// TIA Portal V18 export
FUNCTION "Scale" : Void   // FC2, LAD
{ S7_Optimized_Access := 'TRUE' }
VERSION : 0.1
// stored: AutoNumber true, IsIECCheckEnabled false, SetENOAutomatically false, UDAEnableTagReadback false
   VAR_TEMP
      temp : Real;
   END_VAR
BEGIN

REGION Network 1: Flow meter
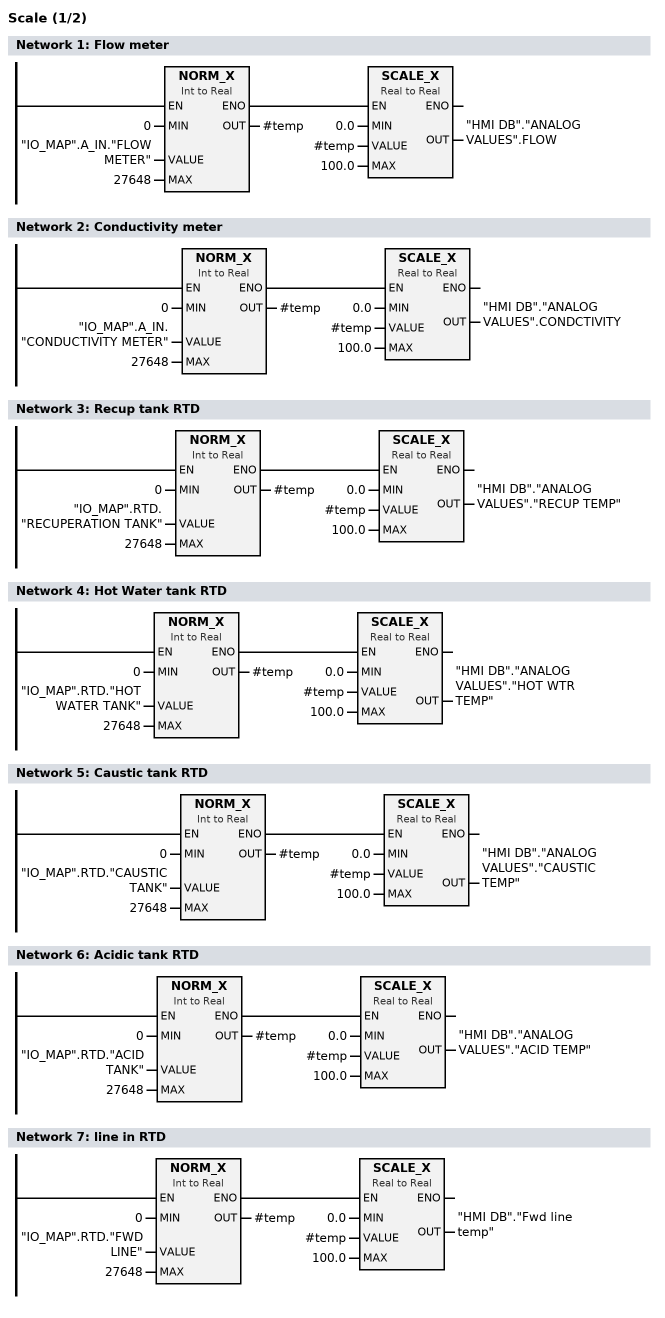
   RUNG wire#powerrail
      { S7_Templates := "[SrcType := Int, DestType := Real]" } Normalize(min := 0, value := "IO_MAP".A_IN."FLOW METER", max := 27648, out => #temp)
      { S7_Templates := "[SrcType := Real, DestType := Real]" } Scale(min := 0.0, value := #temp, max := 100.0, out => "HMI DB"."ANALOG VALUES".FLOW)
   END_RUNG
   // the same network as SCL:
   #temp := NORM_X(MIN := 0, VALUE := "IO_MAP".A_IN."FLOW METER", MAX := 27648);
   "HMI DB"."ANALOG VALUES".FLOW := SCALE_X(MIN := 0.0, VALUE := #temp, MAX := 100.0);
END_REGION

REGION Network 2: Conductivity meter
   RUNG wire#powerrail
      { S7_Templates := "[SrcType := Int, DestType := Real]" } Normalize(min := 0, value := "IO_MAP".A_IN."CONDUCTIVITY METER", max := 27648, out => #temp)
      { S7_Templates := "[SrcType := Real, DestType := Real]" } Scale(min := 0.0, value := #temp, max := 100.0, out => "HMI DB"."ANALOG VALUES".CONDCTIVITY)
   END_RUNG
   // the same network as SCL:
   #temp := NORM_X(MIN := 0, VALUE := "IO_MAP".A_IN."CONDUCTIVITY METER", MAX := 27648);
   "HMI DB"."ANALOG VALUES".CONDCTIVITY := SCALE_X(MIN := 0.0, VALUE := #temp, MAX := 100.0);
END_REGION

REGION Network 3: Recup tank RTD
   RUNG wire#powerrail
      { S7_Templates := "[SrcType := Int, DestType := Real]" } Normalize(min := 0, value := "IO_MAP".RTD."RECUPERATION TANK", max := 27648, out => #temp)
      { S7_Templates := "[SrcType := Real, DestType := Real]" } Scale(min := 0.0, value := #temp, max := 100.0, out => "HMI DB"."ANALOG VALUES"."RECUP TEMP")
   END_RUNG
   // the same network as SCL:
   #temp := NORM_X(MIN := 0, VALUE := "IO_MAP".RTD."RECUPERATION TANK", MAX := 27648);
   "HMI DB"."ANALOG VALUES"."RECUP TEMP" := SCALE_X(MIN := 0.0, VALUE := #temp, MAX := 100.0);
END_REGION

REGION Network 4: Hot Water tank RTD
   RUNG wire#powerrail
      { S7_Templates := "[SrcType := Int, DestType := Real]" } Normalize(min := 0, value := "IO_MAP".RTD."HOT WATER TANK", max := 27648, out => #temp)
      { S7_Templates := "[SrcType := Real, DestType := Real]" } Scale(min := 0.0, value := #temp, max := 100.0, out => "HMI DB"."ANALOG VALUES"."HOT WTR TEMP")
   END_RUNG
   // the same network as SCL:
   #temp := NORM_X(MIN := 0, VALUE := "IO_MAP".RTD."HOT WATER TANK", MAX := 27648);
   "HMI DB"."ANALOG VALUES"."HOT WTR TEMP" := SCALE_X(MIN := 0.0, VALUE := #temp, MAX := 100.0);
END_REGION

REGION Network 5: Caustic tank RTD
   RUNG wire#powerrail
      { S7_Templates := "[SrcType := Int, DestType := Real]" } Normalize(min := 0, value := "IO_MAP".RTD."CAUSTIC TANK", max := 27648, out => #temp)
      { S7_Templates := "[SrcType := Real, DestType := Real]" } Scale(min := 0.0, value := #temp, max := 100.0, out => "HMI DB"."ANALOG VALUES"."CAUSTIC TEMP")
   END_RUNG
   // the same network as SCL:
   #temp := NORM_X(MIN := 0, VALUE := "IO_MAP".RTD."CAUSTIC TANK", MAX := 27648);
   "HMI DB"."ANALOG VALUES"."CAUSTIC TEMP" := SCALE_X(MIN := 0.0, VALUE := #temp, MAX := 100.0);
END_REGION

REGION Network 6: Acidic tank RTD
   RUNG wire#powerrail
      { S7_Templates := "[SrcType := Int, DestType := Real]" } Normalize(min := 0, value := "IO_MAP".RTD."ACID TANK", max := 27648, out => #temp)
      { S7_Templates := "[SrcType := Real, DestType := Real]" } Scale(min := 0.0, value := #temp, max := 100.0, out => "HMI DB"."ANALOG VALUES"."ACID TEMP")
   END_RUNG
   // the same network as SCL:
   #temp := NORM_X(MIN := 0, VALUE := "IO_MAP".RTD."ACID TANK", MAX := 27648);
   "HMI DB"."ANALOG VALUES"."ACID TEMP" := SCALE_X(MIN := 0.0, VALUE := #temp, MAX := 100.0);
END_REGION

REGION Network 7: line in RTD
   RUNG wire#powerrail
      { S7_Templates := "[SrcType := Int, DestType := Real]" } Normalize(min := 0, value := "IO_MAP".RTD."FWD LINE", max := 27648, out => #temp)
      { S7_Templates := "[SrcType := Real, DestType := Real]" } Scale(min := 0.0, value := #temp, max := 100.0, out => "HMI DB"."Fwd line temp")
   END_RUNG
   // the same network as SCL:
   #temp := NORM_X(MIN := 0, VALUE := "IO_MAP".RTD."FWD LINE", MAX := 27648);
   "HMI DB"."Fwd line temp" := SCALE_X(MIN := 0.0, VALUE := #temp, MAX := 100.0);
END_REGION

REGION Network 8: Return line RTD
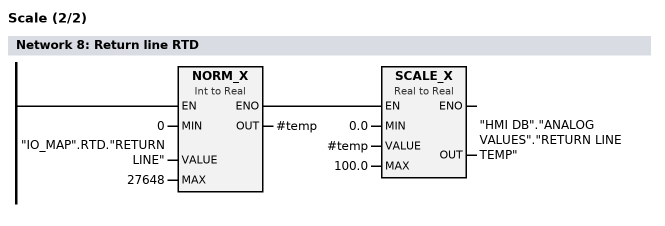
   RUNG wire#powerrail
      { S7_Templates := "[SrcType := Int, DestType := Real]" } Normalize(min := 0, value := "IO_MAP".RTD."RETURN LINE", max := 27648, out => #temp)
      { S7_Templates := "[SrcType := Real, DestType := Real]" } Scale(min := 0.0, value := #temp, max := 100.0, out => "HMI DB"."ANALOG VALUES"."RETURN LINE TEMP")
   END_RUNG
   // the same network as SCL:
   #temp := NORM_X(MIN := 0, VALUE := "IO_MAP".RTD."RETURN LINE", MAX := 27648);
   "HMI DB"."ANALOG VALUES"."RETURN LINE TEMP" := SCALE_X(MIN := 0.0, VALUE := #temp, MAX := 100.0);
END_REGION
END_FUNCTION
